// TIA Portal V17 export
// export: Created 2022-05-04T07:10:39.9588467Z, ExportSetting WithDefaults, DisplayName Totally Integrated Automation Portal, DisplayVersion V17 Update 3, DisplayName TIA Portal Openness, DisplayVersion V17 Update 3, DisplayName TIA Portal Teamcenter Gateway, DisplayVersion V17 Update 3, DisplayName TIA Portal Version Control Interface, DisplayVersion V17, DisplayName SINAMICS Startdrive Advanced, DisplayVersion V17 Update2, DisplayName SINAMICS Startdrive G130, G150, S120, S150, SINAMICS MV, S210, DisplayVersion V17 Update2, DisplayName SINAMICS Startdrive G110M, G120, G120C, G120D, G120P, G115D, DisplayVersion V17 Update2, DisplayName STEP 7 Professional, DisplayVersion V17 Update 3, DisplayName STEP 7 CFC, DisplayVersion V17 Update 1, DisplayName STEP 7 Safety, DisplayVersion V17, DisplayName WinCC UA Professional, DisplayVersion V17 Update 3, DisplayName WinCC Unified Calendar, DisplayVersion V17, DisplayName WinCC Unified Performance Insight, DisplayVersion V17
FUNCTION_BLOCK "Gestion MODBUS TCP CLient"   // FB11, LAD
{ S7_Optimized_Access := 'TRUE' }
VERSION : 0.1
// stored: AutoNumber true, IsIECCheckEnabled false, IsRetainMemResEnabled false, MemoryReserve 100, SetENOAutomatically false, UDAEnableTagReadback false
   VAR
      MB_DATA_ADDR { ExternalAccessible := 'False'; ExternalVisible := 'False'; ExternalWritable := 'False'} : UDInt;
      MB_DATA_LEN { ExternalAccessible := 'False'; ExternalVisible := 'False'; ExternalWritable := 'False'} : UInt := 1;
      MB_DATA_PTR { ExternalAccessible := 'False'; ExternalVisible := 'False'; ExternalWritable := 'False'} : Array[1..1024] of Word;
      MB_CLIENT_Instance { S7_SetPoint := 'True'} : MB_CLIENT;
      CONNECT { S7_SetPoint := 'True'} : TCON_IP_v4;
   END_VAR
   // CONNECT.InterfaceId := 64;
   // CONNECT.ID := 64;
   // CONNECT.ActiveEstablished := true;
   // CONNECT.RemoteAddress.ADDR[1] := 192;
   // CONNECT.RemoteAddress.ADDR[2] := 168;
   // CONNECT.RemoteAddress.ADDR[3] := 0;
   // CONNECT.RemoteAddress.ADDR[4] := 95;
   // CONNECT.RemotePort := 502;
   // CONNECT.LocalPort := 502;
BEGIN

REGION Network 1: Trame Ecriture ' Registre de maintien
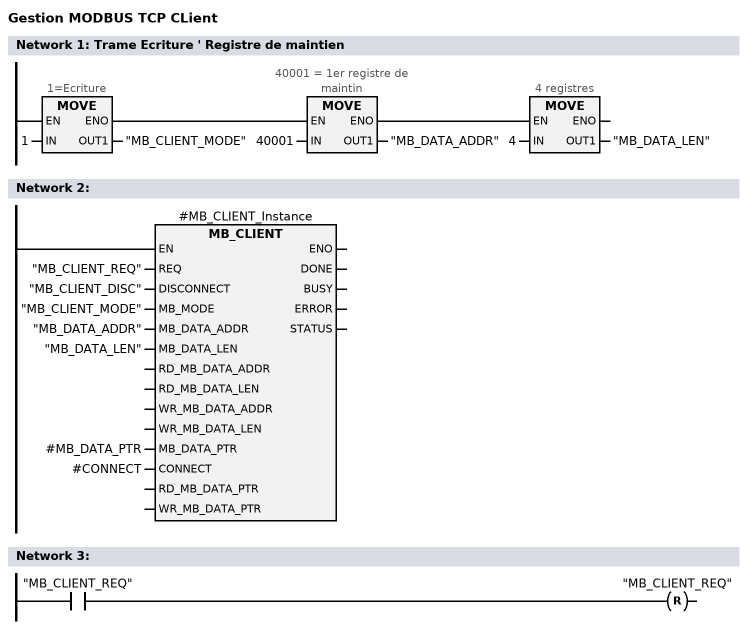
   RUNG wire#powerrail
      Move(in := 1, out1 => "MB_CLIENT_MODE")   // 1=Ecriture
      Move(in := 40001, out1 => "MB_DATA_ADDR")   // 40001 = 1er registre de maintin
      Move(in := 4, out1 => "MB_DATA_LEN")   // 4 registres
   END_RUNG
   // the same network as SCL:
   "MB_CLIENT_MODE" := 1;   // 1=Ecriture
   "MB_DATA_ADDR" := 40001;   // 40001 = 1er registre de maintin
   "MB_DATA_LEN" := 4;   // 4 registres
END_REGION

REGION Network 2
   RUNG wire#powerrail
      #MB_CLIENT_Instance.MB_CLIENT(REQ := "MB_CLIENT_REQ", DISCONNECT := "MB_CLIENT_DISC", MB_MODE := "MB_CLIENT_MODE", MB_DATA_ADDR := "MB_DATA_ADDR", MB_DATA_LEN := "MB_DATA_LEN", RD_MB_DATA_ADDR :=, RD_MB_DATA_LEN :=, WR_MB_DATA_ADDR :=, WR_MB_DATA_LEN :=, MB_DATA_PTR := #MB_DATA_PTR, CONNECT := #CONNECT, RD_MB_DATA_PTR :=, WR_MB_DATA_PTR :=, DONE =>, BUSY =>, ERROR =>, STATUS =>)
   END_RUNG
   // the same network as SCL:
   #MB_CLIENT_Instance(REQ := "MB_CLIENT_REQ",   // MB_CLIENT
                       DISCONNECT := "MB_CLIENT_DISC",
                       MB_MODE := "MB_CLIENT_MODE",
                       MB_DATA_ADDR := "MB_DATA_ADDR",
                       MB_DATA_LEN := "MB_DATA_LEN",
                       MB_DATA_PTR := #MB_DATA_PTR,
                       CONNECT := #CONNECT);
END_REGION

REGION Network 3
   RUNG wire#powerrail
      Contact( "MB_CLIENT_REQ" )
      R_Coil( "MB_CLIENT_REQ" )
   END_RUNG
   // the same network as SCL:
   IF "MB_CLIENT_REQ" THEN "MB_CLIENT_REQ" := FALSE; END_IF;
END_REGION
END_FUNCTION_BLOCK
